RoboDK station: Assistive_UR5e.rdk

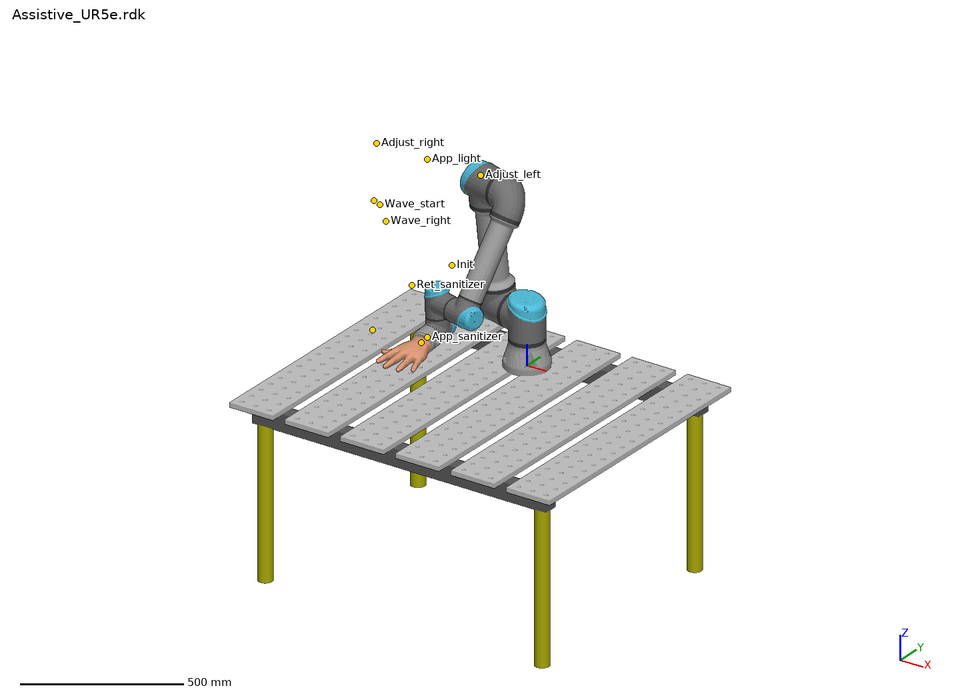
[picture v0: the station drawn from its stored meshes, robots at their saved joint values, targets as dots, program paths as lines]
Station Assistive_UR5e_SW (saved by RoboDK 5.9.2). Poses are relative to the parent item; angles as X-Y-Z fixed-axis rotations.
  - frame UR5e Base at (0, 0, 0) mm
    - robot UR5e: 6 axes, payload 5 kg, reach 850 mm, repeatability 0.03 mm, weight 18.4 kg
        modified DH rows (alpha deg, a mm, theta deg, d mm): 0, 0, 0, 162.5; 90, 0, 180, 0; 0, 425, 0, 0; 0, 392.25, 0, 133.3; -90, 0, 0, 99.7; 90, 0, 180, 99.6
        joint limits [-360, -360, -360, -360, -360, -360] to [360, 360, 360, 360, 360, 360]; home [0, -90, -90, 0, 90, 0]; saved at [-104.807, -96.294, -142.95, 237.206, -109.408, 83.005]
      - tool Hand, TCP at (0, 0, 50) mm, size 54.8 x 155.9 x 193.5 mm, geometry from Hand.stl
    - target Wave_start (Cartesian target) at (-380.86, -238.62, 533.82) mm, rotated rx 0 ry 0 rz 90 deg; joints [-130.679, -89.195, -122.013, 301.208, -90, 130.679] of UR5e
    - target Wave_left (Cartesian target) at (-437.57, -189.83, 513.84) mm, rotated rx -23.64 ry 19.03 rz 85.99 deg; joints [-130.68, -89.19, -122.01, 301.21, -60, 130.68] of UR5e
    - target Wave_right (Cartesian target) at (-324.12, -287.35, 513.84) mm, rotated rx 23.65 ry -19.01 rz 85.98 deg; joints [-130.68, -89.19, -122.01, 301.21, -120, 130.68] of UR5e
  - frame World at (0, 0, 0) mm
    - object Table at (0, 0, 0) mm, size 1193.8 x 965.2 x 609.6 mm, geometry from welding_table.sld
    - target Init (Cartesian target) at (0, -400, 500) mm, rotated rx 90 ry 0 rz 0 deg; joints [-57.836, -65.392, -107.167, 172.559, -57.836, 0] of UR5e
    - target App_sanitizer (Cartesian target) at (-117.86, -360.57, 205.82) mm, rotated rx 6.46 ry -74.9 rz 85.05 deg; joints [28.041, 81.283, -141.189, 208.743, -30.011, 295.899] of UR5e
    - target Press_sanitizer (joint target) at (-117.86, -360.57, 205.82) mm, rotated rx 6.46 ry -74.9 rz 85.05 deg; joints [-87.024, -84.599, -150.631, 250.234, -88.806, 87.94] of UR5e
    - target Ret_sanitizer (Cartesian target) at (-120.86, -440, 413.82) mm, rotated rx 0 ry 0 rz 90 deg; joints [57.655, 34.857, -96.327, 151.47, -90, 302.345] of UR5e
    - target App_light (Cartesian target) at (-119.21, -360.17, 811.64) mm, rotated rx 3.06 ry -61.99 rz 88.16 deg; joints [30.711, -18.437, -87.461, 238.377, -39.477, -51.496] of UR5e
    - target Adjust_left (Cartesian target) at (80.79, -360.17, 811.64) mm, rotated rx 43.07 ry -57.15 rz 21.41 deg; joints [-30.686, -156.981, 77.227, 327.55, -334.661, 180.512] of UR5e
    - target Adjust_right (Cartesian target) at (-309.22, -360.17, 811.64) mm, rotated rx -25.7 ry -50.4 rz 144.98 deg; joints [16.851, -30.17, -38.202, 149.711, -35.518, 30.335] of UR5e
    - target Pick_drug (Cartesian target) at (-369.92, -291.62, 133.7) mm, rotated rx -173.54 ry -83.47 rz -91.74 deg; joints [-140.37, -112.335, -119.224, 220.316, -144.61, 81.532] of UR5e
    - target Move_Drug (Cartesian target) at (-183.13, -300.7, 144.88) mm, rotated rx 145.59 ry -87.67 rz -50.96 deg; joints [-109.51, -91.672, -147.775, 237.341, -114.107, 87.822] of UR5e
    - target Drop_drug (Cartesian target) at (-183.13, -300.7, 144.88) mm, rotated rx -93.07 ry -51.28 rz -172.99 deg; joints [-109.51, -91.672, -147.775, 237.341, -114.107, 127.822] of UR5e
    - target Mix_solution (joint target) at (-183.13, -300.7, 144.88) mm, rotated rx 106.96 ry -83.4 rz -12.25 deg; joints [-109.51, -91.672, -147.775, 237.341, -114.107, 82.822] of UR5e
  - program Init (3 instructions, listed below)
  - program MainProgram (2 instructions, listed below)

--- program Init (robot UR5e) ---
  Est. Ref.: UR5e Base
  Est. herr: Hand
  MoveJ (Init)

--- program MainProgram (robot UR5e) ---
  Llamar Init
  Llamar Init
